PROGRAM MAIN
VAR
	actions : (idle, clear_all, enable_all, disable_all,read_ncyl,read_alias,read_gains,write_gains,read_file,send_waveform_cmd, send_waveform_pwm);
	slave_pos : UINT := 1001;	
	clearfault : FB_ClearFault;
	readncyl : FB_ReadNcyl;
	readalias : FB_ReadAlias;
	readfile : FB_readtextfile;
	waveform_pwm : FB_WritePWM;
	state : INT := 2;
	step : DWORD :=0;
	bError : BOOL;
	t_index : UINT :=1;
	alias : UDINT;
	ncyl: UINT;
	signal : ARRAY[1..60000] OF REAL;
	db : REAL :=14.0;
	dbi : REAL := 0;
	pwm : REAL := 0.0;
	value : REAL := 0.0;
	
	sdo_address: UINT;
	subIndex: BYTE;
	sNetId_local : T_AmsNetId := '10.10.16.19.2.1';	// Address of this computer 
	
// heartbeat
	msthb AT %Q* : UDINT;
	enable AT %Q* : BOOL;
	close_loop AT %Q* : BOOL;
	sp_x AT %Q* : REAL;
	sp_y AT %Q* : REAL;
	sp_z AT %Q* : REAL;
	rb_x AT %I* : REAL;
	rb_y AT %I* : REAL;
	rb_z AT %I* : REAL;
	spr_x AT %I* : REAL;
	spr_y AT %I* : REAL;
	spr_z AT %I* : REAL;
	pwm1 AT %I* : REAL;
	pwm2 AT %I* : REAL;
	pwm3 AT %I* : REAL;
	
	err_mhb AT %I* : BOOL;
	err_f_minmax AT %I* : BOOL;
	err_f_step AT %I* : BOOL;
	err_cal AT %I* : BOOL;
	err_dongle AT %I* : BOOL;
	err_locid AT %I* : BOOL;
	err_soc AT %I* : BOOL;
	err_ff AT %I* : BOOL; 
END_VAR

// send heartbeat to all SA and EPHS

msthb := msthb + 1;


CASE actions OF
	idle:
		state := 2;
		bError := 0;
		t_index := 1;
		sp_x := 0;
		sp_y := 0;
		sp_z := 0;
		
	enable_all :
		enable := TRUE;
		close_loop := TRUE;
		
	disable_all:
		enable := FALSE;
		close_loop := FALSE;
		
	clear_all:
	clearfault(bExecute := TRUE, slv_addr := slave_pos, state => state, bError=> bError );
	IF state = 0 THEN
		actions := idle;
	END_IF
		
	read_ncyl :
		readncyl(bExecute := TRUE, slv_addr := slave_pos, state => state, bError=> bError, value =>ncyl );
		IF state = 0 THEN
			actions := idle;
		END_IF
		
	read_alias :
		readalias(bExecute := TRUE, slv_addr := slave_pos, state => state, bError=> bError, value =>alias );
		IF state = 0 THEN
			actions := idle;
		END_IF
		
	read_file :
		readfile(bread := TRUE,output=>signal,step=>step);
		IF step = 0 THEN
			actions := idle;
		END_IF	
		
	send_waveform_cmd :
	    sp_x := signal[t_index];
		t_index := t_index+1;
		IF t_index>60000 THEN
			t_index := 1;
		END_IF
	
	send_waveform_pwm:
		waveform_pwm(bExecute := TRUE, slv_addr := slave_pos,value :=  6*signal[t_index], state => state, bError=> bError );
		t_index := t_index+1;
		IF t_index>60000 THEN
			t_index := 1;
		END_IF
END_CASE

END_PROGRAM

(* stored: Version 1.1.0.1, ProductVersion 3.1.4024.9
   POU MAIN: Id {59180f09-19c6-4522-85fb-df79ccf53613}, SpecialFunc None *)
